Staubli VAL3: page_pallet.dtx

TrajPallet tTrajPallet
  [0]
    TrajPointItem tData
      [0]
        TrajectoryItem tSuper
          [0]
            num distance
            num moveType
            num nTime
            num nStop
            num nTcpAction
            string comment
            bool toStop
            mdesc nom_speed = {tmax=300, rmax=9999, leave=30, reach=30}
            InstrItem iInstr[3]
              [0]
                string sType
                string sData
              [1]
                string sType
                string sData
              [2]
                string sType
                string sData
            num nMoveId
        pointRx pPoint = {fatherId=tTrajPallet[0].fFrame[0]}
        num nType
    frame fFrame = {fatherId=tTrajPallet[0].fReference[0]}
    num nIndexTool
    string sID
    trsf trAppro[2]
      [0] = {z=-50}
      [1] = {z=-50}
    trsf trDepart[2]
      [0] = {z=-50}
      [1] = {z=-50}
    num nX = 1
    num nY = 1
    num nZ = 1
    num nIndex = 1
    num nDistanceXYZ[3]
      [0] = 1
      [1] = 1
      [2] = 1
    string sAction
    pointRx pO = {fatherId=tTrajPallet[0].fReference[0]}
    pointRx pX = {fatherId=tTrajPallet[0].fReference[0]}
    pointRx pY = {fatherId=tTrajPallet[0].fReference[0]}
    pointRx pZ = {fatherId=tTrajPallet[0].fReference[0]}
    num nSpeedApproach = 300
    num nSpeedDepart = 300
    num nIndexFrame
    frame fReference = {fatherId=world[0]}
bool bButton[8]
  [1] = true
  [4] = true
  [5] = true
  [6] = true
  [7] = true
bool bExit
bool bLarge
bool bOnActionLine
bool bToSave
num nIndex
num nKey = -1
num nPosition = 1
num nRefresh
num nTime = 2
pointRx pNull = {fatherId=world[0]}
pointRx pO = {fatherId=world[0]}
pointRx pOrigin = {fatherId=world[0]}
string sAction
string sEvent = "on Layer 1>"
public string sItems = "test"
string sList[8]
  [0] = "position > 2/1"
  [1] = "pos.  X  > 1/1"
  [2] = "pos.  Y  > 1/1"
  [3] = "pos.  Z  > 2/1"
  [4] = "  dX     > 1  "
  [5] = "  dY     > 1  "
  [6] = "  dZ     > 1  "
  [7] = "on Layer 1>"
string sMenu[8]
  [1] = "Edit Pallet"
  [4] = "Wizard"
  [5] = "Reset"
  [6] = "Back"
  [7] = "Next"
string sPalletName = "test"
num nView
frame fFather = {fatherId=world[0]}
